{attribute 'qualified_only'}
VAR_GLOBAL
	axis_a : AXIS_REF;
END_VAR

(* stored: Version 1.1.0.1, ProductVersion 3.1.4024.12
   GVL GVL: Id {adb180d6-b4d0-4e56-98e1-2b7d940c1ea2} *)
